(* IEC 61131-3 sources: volt/packages/volt-lsp-iec/test-corpus/pro2193/Device/Plc Logic/Application/99 Library/Function Blocks/Pnoz Alarms, 6 files *)

(* ---- PnozAlarmsBaseFB.pou ---- *)
{attribute 'reflection'}
{attribute 'symbol' := 'none'}
FUNCTION_BLOCK PUBLIC ABSTRACT PnozAlarmsBaseFB
VAR_INPUT
	elementId					: UINT;							// Element id of source in Pnozmulti Configurator
	ModuleParent				: L_IMHP.L_IMHP_IModuleHandler;
END_VAR
VAR_OUTPUT
	ModuleHandler				: L_IMHP.L_IMHP_ModuleHandler;	// Lenze module handler (No need to call this FB)
END_VAR
VAR
	{attribute 'instance-path'}
	{attribute 'noinit'}
	{attribute 'hide'}
	_instanceName				: STRING(80);		// Private backing field for instance name (automatically generated by compiler)
END_VAR

%LANGUAGE ST
Initialize();

END_FUNCTION_BLOCK

METHOD PRIVATE Initialize
VAR_INST
	{attribute 'init_on_onlchange' }
	initialized	: BOOL;
END_VAR

%LANGUAGE ST
IF initialized THEN
	RETURN;
END_IF

ParseInstanceName(ADR(_instanceName));

ModuleHandler.CompName	:= InstanceName;
ModuleHandler.Layer		:= L_IMHP_Layer.Tech_Application;
ModuleHandler.CompType	:= L_IMHP_ComponentType.GeneralMachineModule;

// Warning: Only when module is of CompType = MachineModule or GeneralMachineModule, are active alarms kicked up to the parent module!

ModuleHandler.SetParent(
					ModuleHandlerParent	:= ModuleParent,
					RelationShip		:= L_IMHP.L_IMHP_RelationshipID.ApplicationView);

initialized := TRUE;

END_METHOD

// Automatically generated name of the instance
{attribute 'monitoring':='call'}
PROPERTY PUBLIC InstanceName : STRING(80)

GET
VAR
END_VAR

%LANGUAGE ST
InstanceName := _instanceName;

END_GET
END_PROPERTY

(* ---- PnozEmergencyStopAlarmsFB.pou ---- *)
// Throw error messages when a emergency stop is pressed
FUNCTION_BLOCK PnozEmergencyStopAlarmsFB
EXTENDS PnozAlarmsBaseFB
VAR_INPUT
	eStopOperated			: BOOL;		// E-STOP pushbutton was operated (bit 1)
	contactFailed			: BOOL;		// N/C contact 1 or 2 failed to switch or switched too late (bit 5)
	errorTestPulse			: BOOL;		// Error in the test pulse wiring (bit 8)
END_VAR
VAR
	eStopOperatedAlarm		: SetErrorFB;
	contactFailedAlarm		: SetErrorFB;
	errorTestPulseAlarm		: SetErrorFB;
END_VAR

%LANGUAGE ST
SUPER^();

eStopOperatedAlarm(
	moduleHandler	:= ModuleHandler,
	textRefId		:= Pnoz_Errors,
	errorId			:= 1,		// E-STOP pushbutton is operated.
	alarmCondition	:= eStopOperated,
	alarmDelay		:= 0.0,
	severity		:= enumErrorSeverity.Warning,
	reaction		:= enumErrorReaction.No_reaction);

contactFailedAlarm(
	moduleHandler	:= ModuleHandler,
	textRefId		:= Pnoz_Errors,
	errorId			:= 2,		// N/C contact 1 or 2 failed to switch or switched too late
	alarmCondition	:= contactFailed,
	alarmDelay		:= 0.0,
	severity		:= enumErrorSeverity.Fault,
	reaction		:= enumErrorReaction.No_reaction,
	active			=> );

errorTestPulseAlarm(
	moduleHandler	:= ModuleHandler,
	textRefId		:= Pnoz_Errors,
	errorId			:= 3,		// Error in the test pulse wiring
	alarmCondition	:= errorTestPulse,
	alarmDelay		:= 0.0,
	severity		:= enumErrorSeverity.Fault,
	reaction		:= enumErrorReaction.No_reaction,
	active			=> );

END_FUNCTION_BLOCK

(* ---- PnozEnableSwitchAlarmsFB.pou ---- *)
// Throw error messages when a general input has a problem
FUNCTION_BLOCK PnozEnableSwitchAlarmsFB
EXTENDS PnozAlarmsBaseFB
VAR_INPUT
	switchEnabled			: BOOL;		// Enable switch has not been operated or is fully depressed (signal inverted) (bit 1)
	contactFailed			: BOOL;		// N/C contact 1 or 2 failed to switch or switched too late (bit 5)
	errorTestPulse			: BOOL;		// Error in the test pulse wiring (bit 8)
END_VAR
VAR_OUTPUT
	switchEnabledOut		: BOOL;
END_VAR
VAR
	contactFailedAlarm		: SetErrorFB;
	errorTestPulseAlarm		: SetErrorFB;
END_VAR

%LANGUAGE ST
SUPER^();

switchEnabledOut := switchEnabled;

contactFailedAlarm(
	moduleHandler	:= ModuleHandler,
	textRefId		:= Pnoz_Errors,
	errorId			:= 2,		// N/C contact 1 or 2 failed to switch or switched too late
	alarmCondition	:= contactFailed,
	alarmDelay		:= 0.0,
	severity		:= enumErrorSeverity.Fault,
	reaction		:= enumErrorReaction.No_reaction,
	active			=> );

errorTestPulseAlarm(
	moduleHandler	:= ModuleHandler,
	textRefId		:= Pnoz_Errors,
	errorId			:= 3,		// Error in the test pulse wiring
	alarmCondition	:= errorTestPulse,
	alarmDelay		:= 0.0,
	severity		:= enumErrorSeverity.Fault,
	reaction		:= enumErrorReaction.No_reaction,
	active			=> );

END_FUNCTION_BLOCK

(* ---- PnozOutputWithFeedbackLoopAlarmsFB.pou ---- *)
// Throw error messages when a general output has a problem
FUNCTION_BLOCK PnozOutputWithFeedbackLoopAlarmsFB
EXTENDS PnozAlarmsBaseFB
VAR_INPUT
	feedbackLoopError		: BOOL;		// Feedback loop monitoring is registering an error (bit 8)
END_VAR
VAR
	feedbackLoopErrorAlarm	: SetErrorFB;
END_VAR

%LANGUAGE ST
SUPER^();

feedbackLoopErrorAlarm(
	moduleHandler	:= ModuleHandler,
	textRefId		:= Pnoz_Errors,
	errorId			:= 4,		// Feedback loop monitoring is registering an error
	alarmCondition	:= feedbackLoopError,
	alarmDelay		:= 0.0,
	severity		:= enumErrorSeverity.Fault,
	reaction		:= enumErrorReaction.No_reaction,
	active			=> );

END_FUNCTION_BLOCK

(* ---- PnozSafetyGateAlarmsFB.pou ---- *)
// Throw error messages for safety gates
FUNCTION_BLOCK PnozSafetyGateAlarmsFB
EXTENDS PnozAlarmsBaseFB
VAR_INPUT
	gateOpened				: BOOL;		// Safety gate was opened (bit 1)
	functionTest			: BOOL;		// Function test must be performed (bit 3)
	contactFailed			: BOOL;		// N/C contact 1 or 2 failed to switch or switched too late (bit 5)
	errorTestPulse			: BOOL;		// Error in the test pulse wiring (bit 8)
END_VAR
VAR_OUTPUT
	gateOpenedOut			: BOOL;
END_VAR
VAR
	functionTestAlarm		: SetErrorFB;
	contactFailedAlarm		: SetErrorFB;
	errorTestPulseAlarm		: SetErrorFB;
END_VAR

%LANGUAGE ST
SUPER^();

gateOpenedOut := gateOpened;

functionTestAlarm(
	moduleHandler	:= ModuleHandler,
	textRefId		:= Pnoz_Errors,
	errorId			:= 5,		// Function test must be performed
	alarmCondition	:= functionTest,
	alarmDelay		:= 0.0,
	severity		:= enumErrorSeverity.Warning,
	reaction		:= enumErrorReaction.No_reaction);

contactFailedAlarm(
	moduleHandler	:= ModuleHandler,
	textRefId		:= Pnoz_Errors,
	errorId			:= 2,		// N/C contact 1 or 2 failed to switch or switched too late
	alarmCondition	:= contactFailed,
	alarmDelay		:= 0.0,
	severity		:= enumErrorSeverity.Fault,
	reaction		:= enumErrorReaction.No_reaction,
	active			=> );

errorTestPulseAlarm(
	moduleHandler	:= ModuleHandler,
	textRefId		:= Pnoz_Errors,
	errorId			:= 3,		// Error in the test pulse wiring
	alarmCondition	:= errorTestPulse,
	alarmDelay		:= 0.0,
	severity		:= enumErrorSeverity.Fault,
	reaction		:= enumErrorReaction.No_reaction,
	active			=> );

END_FUNCTION_BLOCK

(* ---- PnozSafetyMatAlarmsFB.pou ---- *)
// Throw error messages when a emergency stop is pressed
FUNCTION_BLOCK PnozSafetyMatAlarmsFB
EXTENDS PnozAlarmsBaseFB
VAR_INPUT
	activated				: BOOL;		// Safety mat was activated (bit 1)
	readyForReset			: BOOL;		// Safety mat is ready for reset (bit 2)
	error					: BOOL;		// Error caused by safety mat (bit 5)
END_VAR
VAR
	activatedAlarm			: SetErrorFB;
	readyForResetAlarm		: SetErrorFB;
	errorAlarm				: SetErrorFB;
END_VAR

%LANGUAGE ST
SUPER^();

activatedAlarm(
	moduleHandler	:= ModuleHandler,
	textRefId		:= Pnoz_Errors,
	errorId			:= 6,		// Safety mat was activated
	alarmCondition	:= activated,
	alarmDelay		:= 0.0,
	severity		:= enumErrorSeverity.Fault,
	reaction		:= enumErrorReaction.Stop);

readyForResetAlarm(
	moduleHandler	:= ModuleHandler,
	textRefId		:= Pnoz_Errors,
	errorId			:= 7,		// Safety mat is ready for reset
	alarmCondition	:= readyForReset,
	alarmDelay		:= 0.0,
	severity		:= enumErrorSeverity.Information,
	reaction		:= enumErrorReaction.No_reaction,
	active			=> );

errorAlarm(
	moduleHandler	:= ModuleHandler,
	textRefId		:= Pnoz_Errors,
	errorId			:= 8,		// Error caused by safety mat
	alarmCondition	:= error,
	alarmDelay		:= 0.0,
	severity		:= enumErrorSeverity.Fault,
	reaction		:= enumErrorReaction.No_reaction,
	active			=> );

END_FUNCTION_BLOCK
